{attribute 'GeneratedUsingTerminal: EL2622-0010-0016'}
{attribute addProperty BoxType "EL2622-0010-0016"}
{attribute addProperty Id "InputsAT %I*Inputs_298FB92D1Channel_1AT %Q*Channel_42CA91F71Channel_2AT %Q*Channel_42CA91F71WcStateAT %I*WcState_9091E0EB2InfoDataAT %I*InfoData_6F19DB2B2"}
{attribute addProperty CRC "1206271783"}
{attribute addProperty Size "7"}
TYPE EL2622_47E63F27 EXTENDS EtcSlaveTerminalBase_947E5A46 :
STRUCT
	{attribute addProperty Name "Inputs"}
	Inputs : Inputs_298FB92D;
	{attribute addProperty Name "Channel_1"}
	Channel_1 : Channel_42CA91F7;
	{attribute addProperty Name "Channel_2"}
	Channel_2 : Channel_42CA91F7;
	{attribute addProperty Name "WcState"}
	WcState : WcState_9091E0EB;
	{attribute addProperty Name "InfoData"}
	InfoData : InfoData_6F19DB2B;
END_STRUCT
END_TYPE

(* stored: Version 1.2.0.0, ProductVersion 3.1.4024.9
   DUT EL2622_47E63F27: Id {86fed093-9026-445c-83c7-cc6456712f50} *)
